Yaskawa INFORM job: MT_BIN.JBI

/JOB
//NAME MT_BIN
//POS
///NPOS 4,0,0,0,0,0
///TOOL 0
///POSTYPE PULSE
///PULSE
C00000=-365287,68307,203213,143210,135176,-111296
C00001=-367229,160953,197063,138410,139329,-50771
C00002=-365287,68307,203213,143210,135176,-111296
C00003=-206994,4291,120551,103214,157895,-157311
//INST
///DATE 2023/11/30 18:31
///ATTR SC,RW
///GROUP1 RB1
NOP
MOVJ C00000 VJ=50.00 PL=0
MOVL C00001 V=150.0 PL=0
CALL JOB:OPEN_2FG7-1
MOVL C00002 V=500.0 PL=0
MOVJ C00003 VJ=50.00 PL=0
END
